FUNCTION_BLOCK RT_E_TRAIN (* Generation of a finite train of events *)
  (* Description: Copyright (c) 2008 ACIN This program and the accompanying materials are made available under the terms of the Eclipse Public License 2.0 which is available at https://www.eclipse.org/legal/epl-2.0/ SPDX-License-Identifier: EPL-2.0 *)
  (* Version 3.0, 2025-04-14, Patrick Aigner, changed package *)
  (* Version 1.0, 2008-07-10, Alois Zoitl, ACIN *)
  PACKAGE eclipse4diac::rtevents;
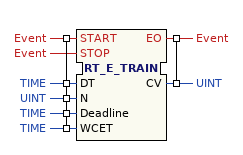
  EVENT_INPUT
    START WITH DT, N, Deadline, WCET;
    STOP;
  END_EVENT
  EVENT_OUTPUT
    EO WITH CV; (* N events at period DT,starting at DT after START *)
  END_EVENT
  VAR_INPUT
    DT : TIME; (* Period between events *)
    N : UINT; (* Number of events to generate *)
    Deadline : TIME;
    WCET : TIME;
  END_VAR
  VAR_OUTPUT
    CV : UINT; (* EO index(0 N-1) *)
  END_VAR
  FBS
    RT_E_CYCLE : eclipse4diac::rtevents::RT_E_CYCLE;
    E_CTU : iec61499::events::E_CTU;
    E_SWITCH : iec61499::events::E_SWITCH;
  END_FBS
  EVENT_CONNECTIONS
    RT_E_CYCLE.EO TO E_CTU.CU;
    START TO E_CTU.R;
    STOP TO RT_E_CYCLE.STOP;
    E_CTU.RO TO RT_E_CYCLE.START;
    E_CTU.CUO TO E_SWITCH.EI;
    E_SWITCH.EO0 TO EO;
    E_SWITCH.EO1 TO RT_E_CYCLE.STOP;
  END_CONNECTIONS
  DATA_CONNECTIONS
    DT TO RT_E_CYCLE.DT;
    Deadline TO RT_E_CYCLE.Deadline;
    WCET TO RT_E_CYCLE.WCET;
    N TO E_CTU.PV;
    E_CTU.CV TO CV;
    E_CTU.Q TO E_SWITCH.G;
  END_CONNECTIONS
END_FUNCTION_BLOCK
